// TwinCAT 3 PLC project Main
// ProgramVersion: 3.1.4022.7
// libraries:
//   Tc2_Standard, * (Beckhoff Automation GmbH)
//   Tc2_System, * (Beckhoff Automation GmbH)
//   Tc3_Module, * (Beckhoff Automation GmbH)
//   VisuSymbols,3.5.10.0,System
// project tree:
//   / GlobalTextList.TcGTLO, PlcTask.TcTTO, Visualization Manager.TcVMO (not stored)
//   GVLs/ TransportSystemIO.TcGVL
//   POUs/ MAIN.TcPOU, DoorControlLogic.TcPOU
// real-time tasks:
//   TASK PlcTask: cycle T#10ms, priority 20, ADS port 350
// I/O:
//   DEVICE Device 2 (CX-BK)
//     Box 1 (CX-BK)
// variable links:
//   Main/Main Instance <-> Device 2 (CX-BK)/Box 1 (CX-BK)
//     PlcTask Inputs/DoorControlLogic.chart_cssd_door_Closed_Signal <-> Term 2 (KL1184)/Channel 1/Input
//     PlcTask Inputs/DoorControlLogic.chart_cssd_door_Opened_Signal <-> Term 3 (KL1184)/Channel 1/Input
//     PlcTask Outputs/DoorControlLogic.chart_cssd_door_Contact <-> Term 5 (KL2622)/Channel 1/Output
//     PlcTask Outputs/DoorControlLogic.chart_cssd_door_Hold <-> Term 4 (KL2622)/Channel 1/Output

CONFIGURATION Main
    RESOURCE PLC ON TwinCAT3
        TASK PlcTask(INTERVAL := T#10ms, PRIORITY := 20);
        PROGRAM MAIN WITH PlcTask : MAIN;
    END_RESOURCE
END_CONFIGURATION

// ---- GVLs/TransportSystemIO.TcGVL
{attribute 'qualified_only'}
VAR_GLOBAL

END_VAR

// ---- POUs/MAIN.TcPOU
PROGRAM MAIN
VAR
END_VAR

DoorControlLogic();

END_PROGRAM

// ---- POUs/DoorControlLogic.TcPOU
PROGRAM DoorControlLogic
VAR
	{attribute 'OPC.UA.DA' := '1'}	
	chart_cssd_door_Status						:	BOOL;	// Status of door contact - True:Open | False:Close
	
	{attribute 'OPC.UA.DA' := '1'}	
	chart_cssd_door_Open_Command	AT %I*		: 	BOOL;	// Open Door 1 command from robot

	{attribute 'OPC.UA.DA' := '1'}			
	chart_cssd_door_Close_Command	AT %I*		:	BOOL	:= FALSE;	// Close Door 1 command from robot, init to be false

	{attribute 'OPC.UA.DA' := '1'}		
	chart_cssd_door_Opened_Signal	AT %I*		:	BOOL;
	
	{attribute 'OPC.UA.DA' := '1'}		
	chart_cssd_door_Closed_Signal	AT %I*		: 	BOOL;
	
	{attribute 'OPC.UA.DA' := '1'}		
	chart_cssd_door_Hold			AT %Q*		: 	BOOL;
	
	chart_cssd_door_Contact			AT %Q* 		: 	BOOL	:= FALSE;	// Output to close door contact, init to be false
	
END_VAR

IF chart_cssd_door_Close_Command = TRUE AND NOT chart_cssd_door_Open_Command = TRUE THEN
	chart_cssd_door_Contact := FALSE;
	chart_cssd_door_Hold := FALSE; 
	ELSIF chart_cssd_door_Open_Command = TRUE AND chart_cssd_door_Close_Command = FALSE THEN
		chart_cssd_door_Contact := TRUE;
		chart_cssd_door_Hold := TRUE;		
		ELSIF chart_cssd_door_Open_Command = TRUE AND chart_cssd_door_Close_Command = TRUE THEN
			chart_cssd_door_Contact := FALSE;
			chart_cssd_door_Hold := FALSE;
			chart_cssd_door_Open_Command := FALSE;
			ELSIF chart_cssd_door_Open_Command := FALSE AND chart_cssd_door_Close_Command = FALSE THEN
				chart_cssd_door_Contact := FALSE;
				chart_cssd_door_Hold := FALSE;
				chart_cssd_door_Open_Command := FALSE;
//			ELSIF chart_cssd_door_Open_Command := FALSE AND chart_cssd_door_Close_Command = TRUE THEN
//				chart_cssd_door_Contact := TRUE;
//				chart_cssd_door_Hold := TRUE;
//				chart_cssd_door_Open_Command := TRUE; Commented out as conditions are the same as first condition
	END_IF

IF chart_cssd_door_Opened_Signal = TRUE AND chart_cssd_door_Closed_Signal = FALSE THEN
	chart_cssd_door_Status := TRUE;
	ELSIF chart_cssd_door_Closed_Signal = TRUE AND chart_cssd_door_Opened_Signal = FALSE THEN
		chart_cssd_door_Status := FALSE;
		ELSE
			chart_cssd_door_Status := FALSE;
	END_IF

END_PROGRAM
